(* IEC 61131-3 sources: ATCMcontrol_Engineering/src/TargetBase/Libs/USBManager, 8 files *)

(* ---- Usb_copy.st ---- *)
(*[[
    UserHelpURL= "ATCMfile:Usb_copy.HTML",
]]*)
FUNCTION Usb_copy : UINT
VAR_INPUT
	srcfile : STRING;
	dstfile : STRING;
	src_index : UINT;
	dst_index : UINT;
END_VAR
	INLINE {STDLIB(Usb_copy)}
END_FUNCTION

(* ---- Usb_delete.st ---- *)
(*[[
    UserHelpURL= "ATCMfile:Usb_delete.HTML",
]]*)
FUNCTION Usb_delete : UINT
VAR_INPUT
	file : STRING;
	index : UINT;
END_VAR
	INLINE {STDLIB(Usb_delete)}
END_FUNCTION

(* ---- Usb_diskcopy.st ---- *)
(*[[
    UserHelpURL= "ATCMfile:Usb_diskcopy.HTML",
]]*)
FUNCTION Usb_diskcopy : UINT
VAR_INPUT
	srcfile : STRING;
	dstfile : STRING;
	index : UINT;
END_VAR
	INLINE {STDLIB(Usb_diskcopy)}
END_FUNCTION

(* ---- Usb_feedback.st ---- *)
(*[[
    UserHelpURL= "ATCMfile:Usb_feedback.HTML",
]]*)
FUNCTION Usb_feedback : UINT
VAR_OUTPUT
	USBfeedback : ARRAY[0..2] of INT;
END_VAR
	INLINE {STDLIB(Usb_feedback)}
END_FUNCTION

(* ---- Usb_mkdir.st ---- *)
(*[[
    UserHelpURL= "ATCMfile:Usb_mkdir.HTML",
]]*)
FUNCTION Usb_mkdir : UINT
VAR_INPUT
	dirname : STRING;
	index : UINT;
END_VAR
	INLINE {STDLIB(Usb_mkdir)}
END_FUNCTION

(* ---- Usb_off.st ---- *)
(*[[
    UserHelpURL= "ATCMfile:Usb_off.HTML",
]]*)
FUNCTION Usb_off : UINT
VAR_INPUT
	index : UINT;
END_VAR
	INLINE {STDLIB(Usb_off)}
END_FUNCTION

(* ---- Usb_on.st ---- *)
(*[[
    UserHelpURL= "ATCMfile:Usb_on.HTML",
]]*)
FUNCTION Usb_on : UINT
VAR_INPUT
	index : UINT;
END_VAR
	INLINE {STDLIB(Usb_on)}
END_FUNCTION

(* ---- Usb_status.st ---- *)
(*[[
    UserHelpURL= "ATCMfile:Usb_status.HTML",
]]*)
FUNCTION Usb_status : UINT
VAR_OUTPUT
	USBstatus : ARRAY[0..5] of INT;
END_VAR
	INLINE {STDLIB(Usb_status)}
END_FUNCTION
